FUNCTION_BLOCK FB_ExecutorCutX_Test EXTENDS TcUnit.FB_TestSuite IMPLEMENTS I_GantryConfigProvider
VAR
    Executor : FB_ExecutorCutX;
	Executor_Unhappy     : FB_ExecutorCutX;

    MockCylinder : FB_MockCylinder;
	MockCylinder_Unhappy : FB_MockCylinder;
    MockAxisX    : FB_MockAxis := (Name := 'MockX');
    MockAxisY    : FB_MockAxis := (Name := 'MockY');
    MockAxisZ    : FB_MockAxis := (Name := 'MockZ');
    
    TestRecipe   : FB_RecipeBuilderBorgoWings;
    _TestConfig  : ST_GantryXYZ_Config;
END_VAR

Test_Sequence_ExecutesCutsCorrectly();
Test_Sequence_AbortsOnCylinderError();

PROPERTY Config : ST_GantryXYZ_Config
GET
Config := _TestConfig;
END_GET
SET
_TestConfig := Config;
END_SET
END_PROPERTY

METHOD Test_Sequence_AbortsOnCylinderError
VAR_INST
    Step : INT := 0;
    RecipeConfig : ST_RecipeBuilder_Config;
END_VAR


TEST('Test_Sequence_AbortsOnCylinderError');

Executor_Unhappy.CyclicLogic();

CASE Step OF
    0:
        // 1. ARRANGE - Przygotowanie receptury BorgoWings (6 cięć)
        RecipeConfig.PanelFrontLength := 1000.0;
        TestRecipe.Config := RecipeConfig;
        TestRecipe.Build(); 
		
		_TestConfig.CuttingSpeedX := 10;
		_TestConfig.GroovingSpeedX := 10;
		_TestConfig.RapidSpeedX := 10;
		_TestConfig.CuttingSpeedY := 10;
		_TestConfig.GroovingSpeedY := 10;
		_TestConfig.RapidSpeedY := 10;
	
        
        _TestConfig.CuttingIdleTime := 0.0; 
        
        // ZMUSZAMY MOCK DO AWARII PRZY 3. PRÓBIE WYSUNIĘCIA
        MockCylinder_Unhappy.FailOnExtendCount := 3;
        
        // Wstrzykujemy zależności do Executora "Unhappy"
        Executor_Unhappy.RecipeBuilder  := TestRecipe;
        Executor_Unhappy.ConfigProvider := THIS^; 
        Executor_Unhappy.Cylinder       := MockCylinder_Unhappy;
        Executor_Unhappy.AxisX          := MockAxisX;
        Executor_Unhappy.AxisY          := MockAxisY;
        Executor_Unhappy.AxisZ          := MockAxisZ;
        
        Step := 10;
        
    10:
        // 2. ACT - Start maszyny
        Executor_Unhappy.Execute();
        Step := 20;
        
    20:
        // 3. ASSERT - Oczekujemy BŁĘDU, a nie zakończenia sukcesem!
        IF Executor_Unhappy.Error THEN
            Step := 30; // Sukces testu - Executor wyrzucił błąd
        ELSIF Executor_Unhappy.Done THEN
            AssertTrue(FALSE, 'Cylinder zglosil blad, a Executor zignorowal to i zakonczyl sukcesem!');
            TEST_FINISHED();
        END_IF
        
    30:
        // 4. ASSERT - Weryfikacja dokładnego zachowania podczas awarii
        
        // Oczekujemy, że wysunięcie zostało wywołane dokładnie 3 razy i ani razu więcej
        AssertEquals_INT(Expected := 3, 
                         Actual := MockCylinder_Unhappy.ExtendCallCount, 
                         Message := 'Executor nie zatrzymal sie po bledzie na 3. cieciu!');
                         
        // Oczekujemy, że wsunięcie zostało wywołane tylko 2 razy 
        // (bo przy trzecim wysunięciu był błąd, więc sekwencja spadła z rowerka przed chowaniem!)
        AssertEquals_INT(Expected := 2, 
                         Actual := MockCylinder_Unhappy.RetractCallCount, 
                         Message := 'Bledna liczba wsuniec przed awaria!');
                         
        TEST_FINISHED();
END_CASE
END_METHOD

METHOD Test_Sequence_ExecutesCutsCorrectly
VAR_INST
    Step : INT := 0;
    RecipeConfig : ST_RecipeBuilder_Config;
END_VAR


TEST('Test_Sequence_ExecutesCutsCorrectly');

// Wywołujemy CyclicLogic dla Executora (Mocki nie potrzebują, bo nic w nich w tle nie tyka)
Executor.CyclicLogic();

CASE Step OF
    0:
        // 1. ARRANGE - Przygotowanie receptury Arona (ma 2 cięcia X)
        RecipeConfig.PanelFrontLength := 1000.0;
        TestRecipe.Config := RecipeConfig;
        TestRecipe.Build(); 
		_TestConfig.CuttingSpeedX := 10;
		_TestConfig.GroovingSpeedX := 10;
		_TestConfig.RapidSpeedX := 10;
		_TestConfig.CuttingSpeedY := 10;
		_TestConfig.GroovingSpeedY := 10;
		_TestConfig.RapidSpeedY := 10;
	

        // Czas stabilizacji dla testu ucinamy do zera
        _TestConfig.CuttingIdleTime := 0.0; 
        
        // 2. DEPENDENCY INJECTION - Wstrzykujemy nasze Zaślepki!
        Executor.RecipeBuilder  := TestRecipe;
        Executor.ConfigProvider := THIS^; 
        Executor.Cylinder       := MockCylinder;
        Executor.AxisX          := MockAxisX;
        Executor.AxisY          := MockAxisY;
        Executor.AxisZ          := MockAxisZ;
        
        Step := 10;
        
    10:
        // 3. ACT - Start maszyny
        Executor.Execute();
        Step := 20;
        
    20:
        // 4. Czekamy na koniec sekwencji (dzięki mockom to potrwa ułamki sekund)
        IF Executor.Done THEN
            Step := 30;
        ELSIF Executor.Error THEN
            AssertTrue(FALSE, 'Executor zwrocil Error zamiast Done!');
            TEST_FINISHED();
        END_IF
        
    30:
        // 5. ASSERT - Testujemy Logikę Executora szpiegując Siłownik
        // Arona ma 2 cięcia, więc siłownik musi zostać użyty 2 razy
        AssertEquals_INT(Expected := 6, 
                         Actual := MockCylinder.ExtendCallCount, 
                         Message := 'Bledna liczba wysuniec ostrza!');
                         
        AssertEquals_INT(Expected := 6, 
                         Actual := MockCylinder.RetractCallCount, 
                         Message := 'Bledna liczba wsuniec ostrza!');
                         
        TEST_FINISHED();
END_CASE
END_METHOD

END_FUNCTION_BLOCK

(* stored: Version 1.1.0.1, ProductVersion 3.1.4024.15
   POU FB_ExecutorCutX_Test: Id {7df5cf70-cbe1-43ae-a8be-81dbfb352aaf}, SpecialFunc None
   Property Config: Id {98ba9e04-c6dd-4bd0-953b-b00b87da8f4b}
   Get Get: Id {a7ec6669-d8cc-485f-ad66-71b6c5dd4e2e}
   Set Set: Id {7aa55b37-d946-42cb-bdab-7d5120bef258}
   Method Test_Sequence_AbortsOnCylinderError: Id {9a19ee42-2643-46ec-8532-5c6d8bc6c677}
   Method Test_Sequence_ExecutesCutsCorrectly: Id {c2729daa-46da-4e16-8826-64d5d470ee9f} *)
